TYPE STATE:
    STRUCT
        curTime: REAL;
        dvar_M_hw_button: DINT;
        dvar_M_hw_lamp_bit: BOOL;
        dvar_M_hw_lamp: DINT;
        dvar_M_sup: DINT;
        cvar_M_timer_t: REAL;
        dvar_M_timer: DINT;
    END_STRUCT;
END_TYPE
